TYPE ST_HMI_DataSourceHistInfo : 
STRUCT
	sSPGuid: GUID;
	sAlyFilePath: STRING(255);
	sSourceType: STRING(80);
	sTopic: STRING(255);
	sLayoutID: GUID;
	sAlias: STRING(255);
END_STRUCT
END_TYPE

(* stored: DUT ST_HMI_DataSourceHistInfo: Id c832f19f-a3f6-4abb-b47a-07f954ac21f4 *)
